PROGRAM MAIN
VAR
	Saegeautomat : Saegeautomat;
END_VAR

Saegeautomat();

END_PROGRAM

(* stored: Version 1.1.0.1, ProductVersion 3.1.4024.16
   POU MAIN: Id {14b975ff-daf1-4eb0-a595-be74e665f929}, SpecialFunc None *)
